PROGRAM Events
VAR
	Send_Start_Event : Send_Event_FB;
	Start_Event  : TcEventEntry := TC_Events.Pelletizer_Events.Start_Button_Event;
	
	Send_Stop_Event : Send_Event_FB;
	Stop_Event  : TcEventEntry := TC_Events.Pelletizer_Events.Stop_Button_Event;
//////////////////////////////////////////////////////////////////////////////////////////////////////////////////
	Send_EmergencyStop_Event : Send_Event_FB;
	EmergencyStop_Event : TcEventEntry := TC_Events.Pelletizer_Events.Emergency_Stop_Set_Event;

	Send_EmergencyStop_Reset_Event : Send_Event_FB;
	EmergencyStop_Reset_Event : TcEventEntry := TC_Events.Pelletizer_Events.Emergency_Stop_Reset_Event;
//////////////////////////////////////////////////////////////////////////////////////////////////////////////////	
	Send_Feedroll_Drive_Fault_Event : Send_Event_FB;
	Feedroll_Drive_Fault_Event : TcEventEntry := TC_Events.Pelletizer_Events.Feedroll_Drive_Fault_Event;
	
	Send_Feedroll_Drive_Fault_Reset_Event : Send_Event_FB;
	Feedroll_Drive_Fault_Reset_Event : TcEventEntry := TC_Events.Pelletizer_Events.Feedroll_Drive_Fault_Reset_Event;
//////////////////////////////////////////////////////////////////////////////////////////////////////////////////	
	Send_Rotor_Drive_Fault_Event : Send_Event_FB;
	Rotor_Drive_Fault_Event : TcEventEntry := TC_Events.Pelletizer_Events.Rotor_Drive_Fault_Event;
	
	Send_Rotor_Drive_Fault_Reset_Event : Send_Event_FB;
	Rotor_Drive_Fault_Reset_Event : TcEventEntry := TC_Events.Pelletizer_Events.Rotor_Drive_Fault_Reset_Event;
//////////////////////////////////////////////////////////////////////////////////////////////////////////////////
	Send_Machine_Shutdown_Event : Send_Event_FB;
	Machine_Shutdown_Event : TcEventEntry := TC_Events.Pelletizer_Events.Machine_Shutdown_Event;	
	
	Send_Machine_PowerOn_Event : Send_Event_FB;
	Machine_PowerOn_Event : TcEventEntry := TC_Events.Pelletizer_Events.Machine_PowerOn_Event;
//////////////////////////////////////////////////////////////////////////////////////////////////////////////////	
	Send_Change_Filter_Event : Send_Event_FB;
	Change_Filter_Event : TcEventEntry := TC_Events.AirKnife_Events.Change_Filter_Event;	
	
	Send_Filter_OKAY_Event : Send_Event_FB;
	Filter_OKAY_Event : TcEventEntry := TC_Events.AirKnife_Events.Filter_OKAY_Event;
//////////////////////////////////////////////////////////////////////////////////////////////////////////////////	
	Send_Local_Mode_Active : Send_Event_FB;
	Local_Mode_Active : TcEventEntry := TC_Events.Waterbath_Events.Local_Mode_Active;
	
	Send_Remote_Mode_Active : Send_Event_FB;
	Remote_Mode_Active : TcEventEntry := TC_Events.Waterbath_Events.Remote_Mode_Active;
//////////////////////////////////////////////////////////////////////////////////////////////////////////////////	
	Send_Pump_Start_Event : Send_Event_FB;
	Pump_Start_Event : TcEventEntry := TC_Events.Waterbath_Events.Pump_Start_Event;
	
	Send_Pump_Stop_Event : Send_Event_FB;
	Pump_Stop_Event : TcEventEntry := TC_Events.Waterbath_Events.Pump_Stop_Event;
//////////////////////////////////////////////////////////////////////////////////////////////////////////////////	
	
	First_Scan : BOOL := False;	
END_VAR

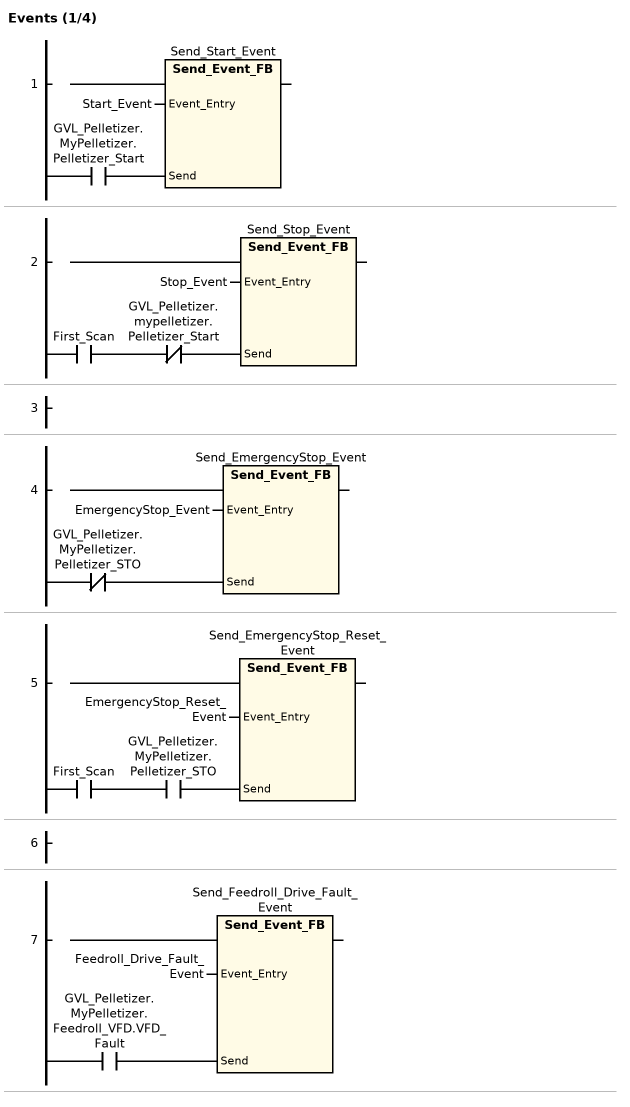
// NETWORK 1
Send_Start_Event(Event_Entry := Start_Event, Send := GVL_Pelletizer.MyPelletizer.Pelletizer_Start); // Send_Event_FB

// NETWORK 2
Send_Stop_Event(Event_Entry := Stop_Event, Send := First_Scan AND NOT GVL_Pelletizer.mypelletizer.Pelletizer_Start); // Send_Event_FB

// NETWORK 3

// NETWORK 4
Send_EmergencyStop_Event(Event_Entry := EmergencyStop_Event, Send := NOT GVL_Pelletizer.MyPelletizer.Pelletizer_STO); // Send_Event_FB

// NETWORK 5
Send_EmergencyStop_Reset_Event(Event_Entry := EmergencyStop_Reset_Event, Send := First_Scan AND GVL_Pelletizer.MyPelletizer.Pelletizer_STO); // Send_Event_FB

// NETWORK 6

// NETWORK 7
Send_Feedroll_Drive_Fault_Event(Event_Entry := Feedroll_Drive_Fault_Event, Send := GVL_Pelletizer.MyPelletizer.Feedroll_VFD.VFD_Fault); // Send_Event_FB

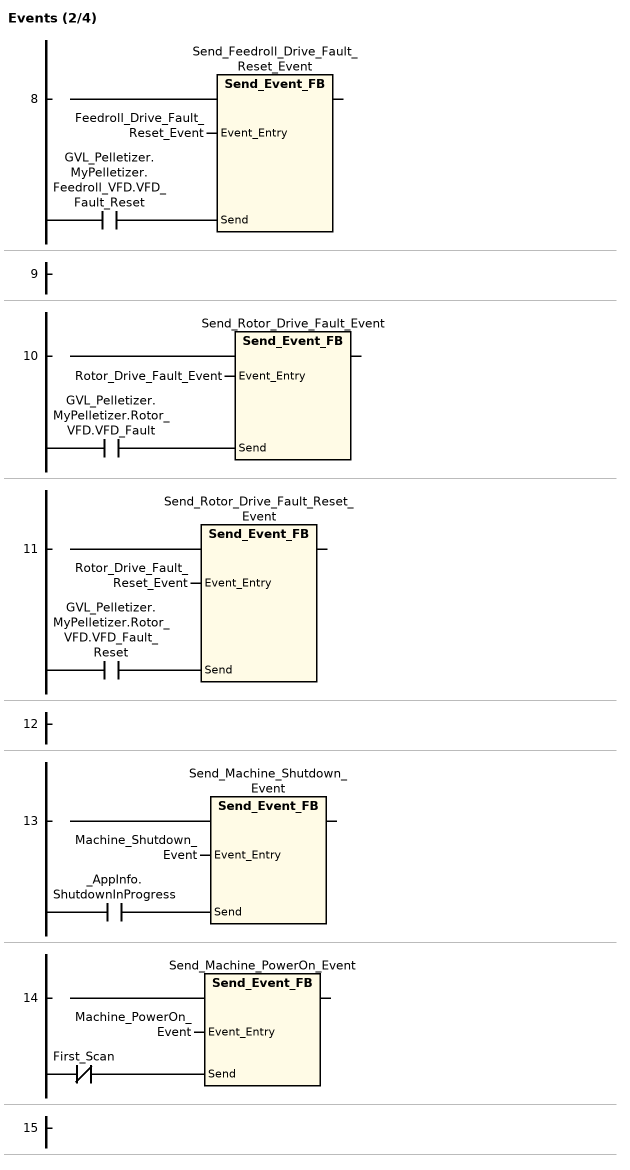
// NETWORK 8
Send_Feedroll_Drive_Fault_Reset_Event(Event_Entry := Feedroll_Drive_Fault_Reset_Event, Send := GVL_Pelletizer.MyPelletizer.Feedroll_VFD.VFD_Fault_Reset); // Send_Event_FB

// NETWORK 9

// NETWORK 10
Send_Rotor_Drive_Fault_Event(Event_Entry := Rotor_Drive_Fault_Event, Send := GVL_Pelletizer.MyPelletizer.Rotor_VFD.VFD_Fault); // Send_Event_FB

// NETWORK 11
Send_Rotor_Drive_Fault_Reset_Event(Event_Entry := Rotor_Drive_Fault_Reset_Event, Send := GVL_Pelletizer.MyPelletizer.Rotor_VFD.VFD_Fault_Reset); // Send_Event_FB

// NETWORK 12

// NETWORK 13
Send_Machine_Shutdown_Event(Event_Entry := Machine_Shutdown_Event, Send := _AppInfo.ShutdownInProgress); // Send_Event_FB

// NETWORK 14
Send_Machine_PowerOn_Event(Event_Entry := Machine_PowerOn_Event, Send := NOT First_Scan); // Send_Event_FB

// NETWORK 15

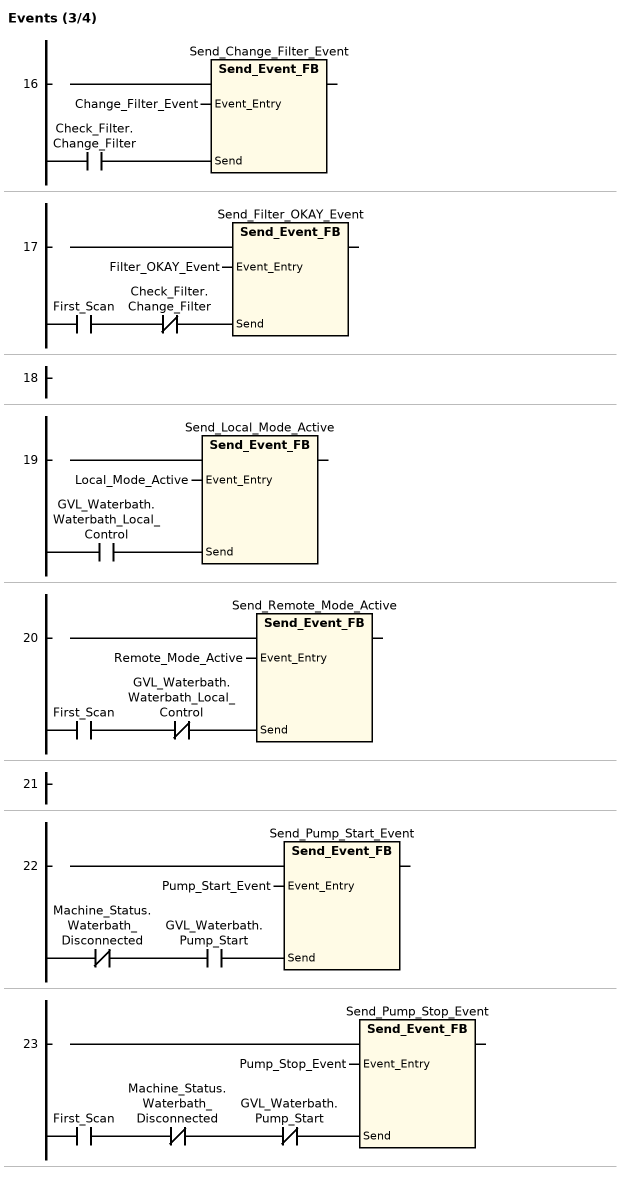
// NETWORK 16
Send_Change_Filter_Event(Event_Entry := Change_Filter_Event, Send := Check_Filter.Change_Filter); // Send_Event_FB

// NETWORK 17
Send_Filter_OKAY_Event(Event_Entry := Filter_OKAY_Event, Send := First_Scan AND NOT Check_Filter.Change_Filter); // Send_Event_FB

// NETWORK 18

// NETWORK 19
Send_Local_Mode_Active(Event_Entry := Local_Mode_Active, Send := GVL_Waterbath.Waterbath_Local_Control); // Send_Event_FB

// NETWORK 20
Send_Remote_Mode_Active(Event_Entry := Remote_Mode_Active, Send := First_Scan AND NOT GVL_Waterbath.Waterbath_Local_Control); // Send_Event_FB

// NETWORK 21

// NETWORK 22
Send_Pump_Start_Event(Event_Entry := Pump_Start_Event, Send := NOT Machine_Status.Waterbath_Disconnected AND GVL_Waterbath.Pump_Start); // Send_Event_FB

// NETWORK 23
Send_Pump_Stop_Event(Event_Entry := Pump_Stop_Event, Send := First_Scan AND NOT Machine_Status.Waterbath_Disconnected AND NOT GVL_Waterbath.Pump_Start); // Send_Event_FB

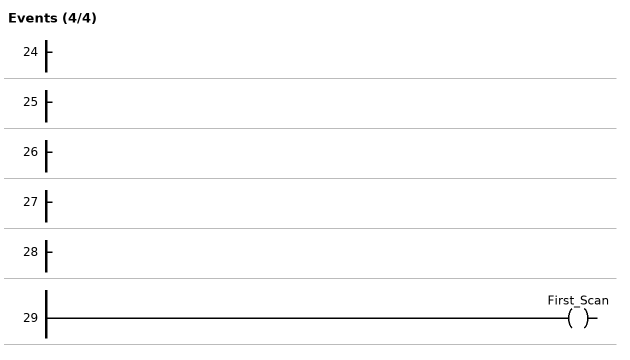
// NETWORK 24

// NETWORK 25

// NETWORK 26

// NETWORK 27

// NETWORK 28

// NETWORK 29
First_Scan := TRUE;

END_PROGRAM

(* stored: Version 1.1.0.1, ProductVersion 3.1.4024.12
   POU Events: Id {bf716019-7947-4d54-948b-ddf8d1322a0f}, SpecialFunc None *)
